// TIA Portal V16 export
// export: Created 2025-12-18T09:30:41.3925776Z, ExportSetting WithDefaults, DisplayName Totally Integrated Automation Portal, DisplayVersion V16, DisplayName TIA Portal Version Control Interface, DisplayVersion V16, DisplayName TIA Portal Openness, DisplayVersion V16, DisplayName STEP 7 Professional, DisplayVersion V16, DisplayName STEP 7 Safety, DisplayVersion V16, DisplayName WinCC Advanced, DisplayVersion V16
DATA_BLOCK "Sequence Data Management_DB"   // DB10
VERSION : 0.1
// stored: AutoNumber true, DBAccessibleFromOPCUA true, InstanceOfName Sequence Data Management, InstanceOfType FB
"Sequence Data Management"
   // VAR
   //    WorkStationList1 : Array[0..9] of DInt;
   //    WorkStationList2 : Array[0..9] of DInt;
   //    WorkStationList3 : Array[0..9] of DInt;
   // END_VAR
BEGIN
END_DATA_BLOCK
